(* CoDeSys 2.3.10.0 project: main.prx *)
(* Libraries: standard.lib 5.6.98 12:03:02, TcBaseBCxx50.lbx 29.3.07 07:21:36, TcSystemBCxx50.lbx 11.2.10 15:45:50 *)

(* Task configuration *)
TASK Standard (PRIORITY := 0, INTERVAL := T#20ms);
	ADS_block();
	MAIN
END_TASK

(* Global variable list: Global_Variables *)
VAR_GLOBAL
	DD1_2 AT%I* : BOOL;
	DD3  AT%I* : BOOL;
	DO1 AT%I* : BOOL;     (*не задействован*)

	DD1_2_var_off: BOOL := FALSE;
	DD1_2_var_on: BOOL := FALSE;
	DD3_var_off: BOOL := FALSE;
	DD3_var_on: BOOL := FALSE;
	delay_DD1_2_off : TIME := T#1m;
	delay_DD3_off : TIME := T#1m;

(***********out relays for landscape lights************)
	Out AT%Q* : ARRAY [1..18] OF BOOL := FALSE;

(***********out relays garage************)
	garage_OG_22_ABB_replacement AT %Q* : BOOL;
	OutLight1 AT%Q* :BOOL;     (*не задействована*)
	OutLight2 AT%Q* :BOOL;     (*не задействована*)
	OutLight3 AT%Q* :BOOL;     (*не задействована*)
	OutLight4 AT%Q* :BOOL;     (*не задействована*)

(***********keypad buttons************)
	UOG18_1 AT%I* : BOOL;	(*Клавиша ручного вкл/выкл освещения гаража в комнате охраны*)
	UOG18_2 AT%I* : BOOL;	(*Клавиша ручного вкл/выкл освещения ландшафта в комнате охраны*)
	UOG18_1_mem : BOOL;	(*положение клавиши предыдущего цикла*)
	UOG18_2_mem : BOOL;	(*положение клавиши предыдущего цикла*)
(***********keypad buttons************)

	KNX_NIGHT : BOOL;
	NIGHT_KNXNET : BOOL;
	NIGHT_KNXNET_FLAG : BOOL;
	NIGHT_CLOCK : BOOL;
	daynightbit : INT := 8;
	SystemTime : TIMESTRUCT;

	KNX_NIGHT_front: BOOL;
	KNX_DAY_front: BOOL := TRUE;
	KNX_GatesLight : BOOL;
	SWAP_CYCLE : BOOL;
	garage_OG_22 : BOOL;

	AdsUdpOutcomingStack : ARRAY [1..19] OF BOOL;
	AdsUdpReceiveStack : ARRAY [1..19] OF BOOL;
	AdsUdpEmptyStack : ARRAY [1..19] OF BOOL := FALSE;
	TESTneeds : BOOL;

	var1 : BOOL;
	var2 : BOOL;
END_VAR

(* Global variable list: TwinCAT_Configuration *)
(* Generated automatically by TwinCAT - (read only) *)
VAR_CONFIG
	.DD1_2 AT %IX8.0 : BOOL;	(*  ~ {LinkedWith:TIID^Device 1 (BX-BK)^BX KBus-Device^Term 2 (KL1408)^Channel 5^Input} *)
	.DD3 AT %IX8.1 : BOOL;	(*  ~ {LinkedWith:TIID^Device 1 (BX-BK)^BX KBus-Device^Term 2 (KL1408)^Channel 7^Input} *)
	.DO1 AT %IX8.2 : BOOL;	(*  ~ {LinkedWith:TIID^Device 1 (BX-BK)^BX KBus-Device^Term 2 (KL1408)^Channel 1^Input} *)
	.Out AT %QB4 : ARRAY [1..18] OF BOOL;
	.garage_OG_22_ABB_replacement AT %QX24.0 : BOOL;
	.OutLight1 AT %QX2.0 : BOOL;	(*  ~ {LinkedWith:TIID^Device 1 (BX-BK)^BX KBus-Device^Term 8 (KM2604)^Channel 3^Output} *)
	.OutLight2 AT %QX2.1 : BOOL;	(*  ~ {LinkedWith:TIID^Device 1 (BX-BK)^BX KBus-Device^Term 8 (KM2604)^Channel 4^Output} *)
	.OutLight3 AT %QX2.2 : BOOL;
	.OutLight4 AT %QX2.3 : BOOL;
	.UOG18_1 AT %IX12.0 : BOOL;	(*  ~ {LinkedWith:TIID^Device 1 (BX-BK)^BX KBus-Device^Term 2 (KL1408)^Channel 4^Input} *)
	.UOG18_2 AT %IX12.1 : BOOL;	(*  ~ {LinkedWith:TIID^Device 1 (BX-BK)^BX KBus-Device^Term 2 (KL1408)^Channel 2^Input} *)
END_VAR

(* POU ADS_block, CFC *)
PROGRAM ADS_block
VAR
	Timer1: TON;
	ADSreadcxbc1: ADSREAD;
	ADSreadcxbc2: ADSREAD;
	ADSwritecxbc1: ADSWRITE;
	ADSreadcxbc3: ADSREAD;
	ADSreadcxbc4: ADSREAD;
	ADSreadcxbc5: ADSREAD;
	ADSreadcxbc6: ADSREAD;
END_VAR
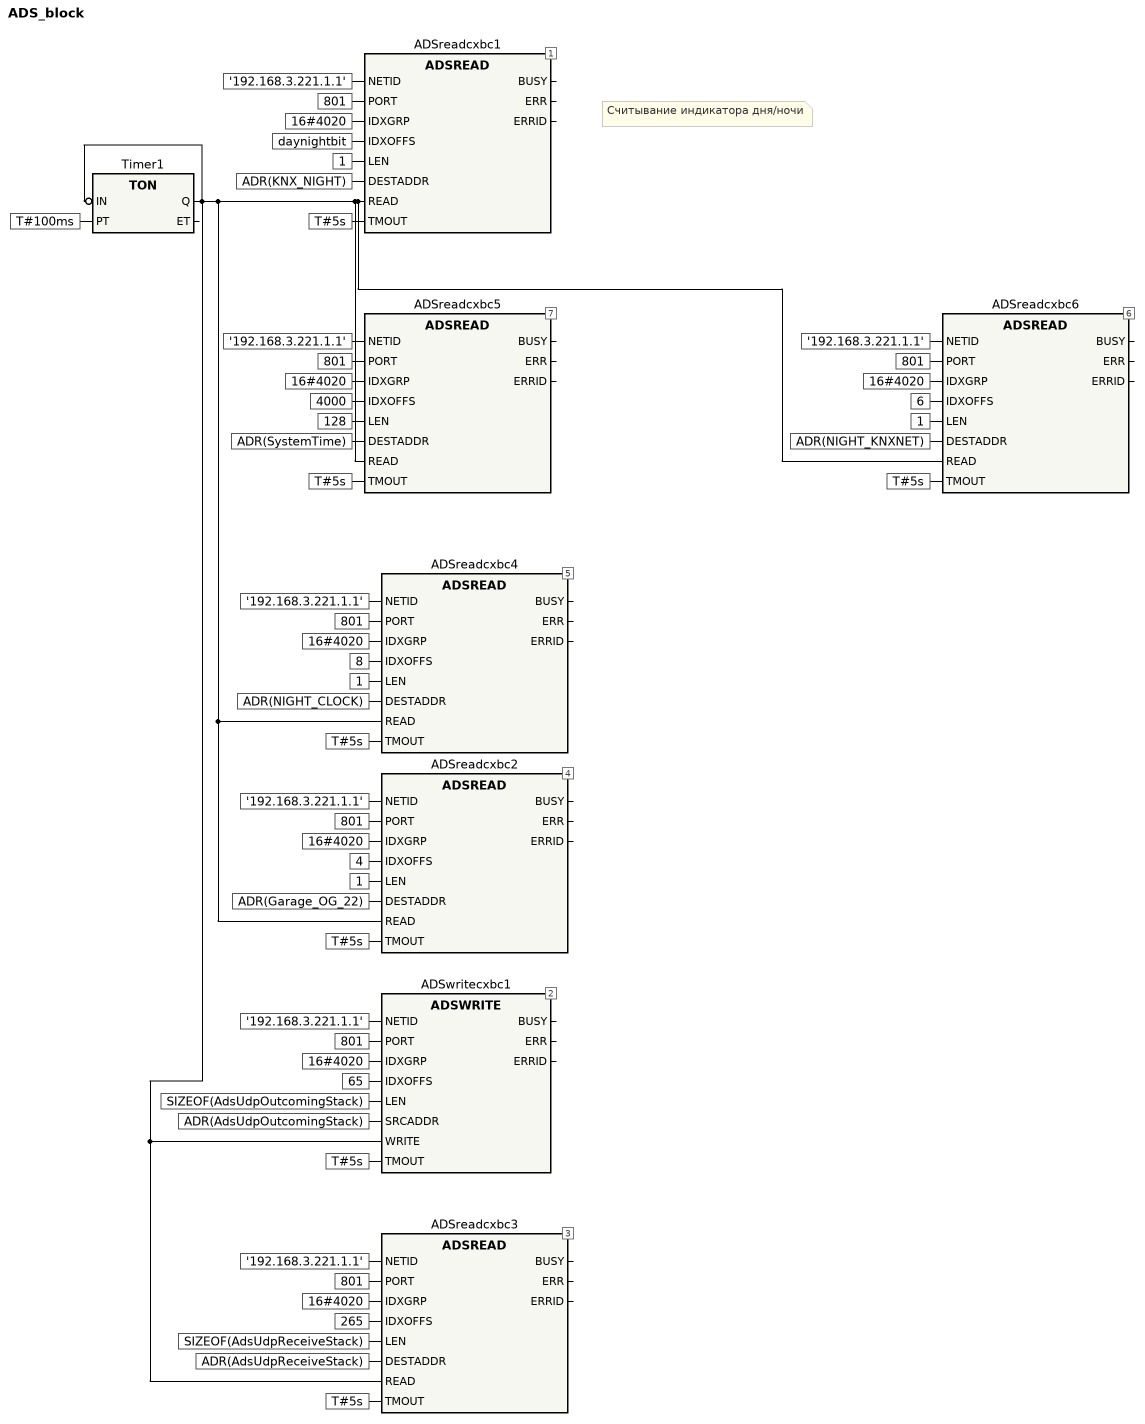
_CFC_ (* Continuous Function Chart, elements in execution order *)
#0 Timer1:TON(IN: NOT #0.Q, PT: T#100ms)
#1 ADSreadcxbc1:ADSREAD(NETID: '192.168.3.221.1.1', PORT: 801, IDXGRP: 16#4020, IDXOFFS: daynightbit, LEN: 1, DESTADDR: ADR(KNX_NIGHT), READ: #0.Q, TMOUT: T#5s)
(* Считывание индикатора дня/ночи *)
#2 ADSwritecxbc1:ADSWRITE(NETID: '192.168.3.221.1.1', PORT: 801, IDXGRP: 16#4020, IDXOFFS: 65, LEN: SIZEOF(AdsUdpOutcomingStack), SRCADDR: ADR(AdsUdpOutcomingStack), WRITE: #0.Q, TMOUT: T#5s)
#3 ADSreadcxbc3:ADSREAD(NETID: '192.168.3.221.1.1', PORT: 801, IDXGRP: 16#4020, IDXOFFS: 265, LEN: SIZEOF(AdsUdpReceiveStack), DESTADDR: ADR(AdsUdpReceiveStack), READ: #0.Q, TMOUT: T#5s)
#4 ADSreadcxbc2:ADSREAD(NETID: '192.168.3.221.1.1', PORT: 801, IDXGRP: 16#4020, IDXOFFS: 4, LEN: 1, DESTADDR: ADR(Garage_OG_22), READ: #0.Q, TMOUT: T#5s)
#5 ADSreadcxbc4:ADSREAD(NETID: '192.168.3.221.1.1', PORT: 801, IDXGRP: 16#4020, IDXOFFS: 8, LEN: 1, DESTADDR: ADR(NIGHT_CLOCK), READ: #0.Q, TMOUT: T#5s)
#6 ADSreadcxbc6:ADSREAD(NETID: '192.168.3.221.1.1', PORT: 801, IDXGRP: 16#4020, IDXOFFS: 6, LEN: 1, DESTADDR: ADR(NIGHT_KNXNET), READ: #0.Q, TMOUT: T#5s)
#7 ADSreadcxbc5:ADSREAD(NETID: '192.168.3.221.1.1', PORT: 801, IDXGRP: 16#4020, IDXOFFS: 4000, LEN: 128, DESTADDR: ADR(SystemTime), READ: #0.Q, TMOUT: T#5s)
_END_CFC_
(* the same logic as Structured Text *)
Timer1(IN := NOT Timer1.Q, PT := T#100ms);
ADSreadcxbc1(NETID := '192.168.3.221.1.1', PORT := 801, IDXGRP := 16#4020, IDXOFFS := daynightbit, LEN := 1, DESTADDR := ADR(KNX_NIGHT), READ := Timer1.Q, TMOUT := T#5s);
(* Считывание индикатора дня/ночи *)
ADSwritecxbc1(NETID := '192.168.3.221.1.1', PORT := 801, IDXGRP := 16#4020, IDXOFFS := 65, LEN := SIZEOF(AdsUdpOutcomingStack), SRCADDR := ADR(AdsUdpOutcomingStack), WRITE := Timer1.Q, TMOUT := T#5s);
ADSreadcxbc3(NETID := '192.168.3.221.1.1', PORT := 801, IDXGRP := 16#4020, IDXOFFS := 265, LEN := SIZEOF(AdsUdpReceiveStack), DESTADDR := ADR(AdsUdpReceiveStack), READ := Timer1.Q, TMOUT := T#5s);
ADSreadcxbc2(NETID := '192.168.3.221.1.1', PORT := 801, IDXGRP := 16#4020, IDXOFFS := 4, LEN := 1, DESTADDR := ADR(Garage_OG_22), READ := Timer1.Q, TMOUT := T#5s);
ADSreadcxbc4(NETID := '192.168.3.221.1.1', PORT := 801, IDXGRP := 16#4020, IDXOFFS := 8, LEN := 1, DESTADDR := ADR(NIGHT_CLOCK), READ := Timer1.Q, TMOUT := T#5s);
ADSreadcxbc6(NETID := '192.168.3.221.1.1', PORT := 801, IDXGRP := 16#4020, IDXOFFS := 6, LEN := 1, DESTADDR := ADR(NIGHT_KNXNET), READ := Timer1.Q, TMOUT := T#5s);
ADSreadcxbc5(NETID := '192.168.3.221.1.1', PORT := 801, IDXGRP := 16#4020, IDXOFFS := 4000, LEN := 128, DESTADDR := ADR(SystemTime), READ := Timer1.Q, TMOUT := T#5s);
END_PROGRAM

(* POU MAIN, ST *)
PROGRAM MAIN
VAR
	i : INT;
	FLAG_I : BOOL := TRUE;
	j: INT;
	Rec_Not_Empty: BOOL;
	k: INT;
	FLAG_01: BOOL;
	HOUR_01: WORD := 2;
	MINUTE_01: WORD := 59;
	HOUR_02: WORD := 10;
	MINUTE_02: WORD := 20;
END_VAR
IF (FLAG_I) THEN (*первый "холостой" цикл, запись положения клавиши ручного вкл/выкл освещения*)
	UOG18_1_mem := UOG18_1;
	UOG18_2_mem := UOG18_2;
	KNX_DAY_front := TRUE;
	FLAG_I := FALSE;
END_IF;

IF (Garage_OG_22) THEN
garage_OG_22_ABB_replacement := TRUE;
ELSE
garage_OG_22_ABB_replacement := FALSE;
END_IF;

IF(UOG18_1 = UOG18_1_mem) THEN; (*вкл/выкл подсветки гаража в комнате охраны*)
ELSE
	Out[5] := NOT(Out[5]);
	Out[6] := NOT(Out[6]);
END_IF;

KNX_night_init; (*подпрограмма получения флага ночь/день по фронтам переменной KNX_NIGHT*)
DD_delay_block; (*подпрограмма обработки сигнала с ДД*)
IF(UOG18_2 = UOG18_2_mem) THEN
		IF (DD1_2_var_on AND DD1_2_var_off = FALSE) THEN   (*Включение/выключение подсветки въезда в гараж от ДД*)
			Out[1] := TRUE;
		END_IF;
		IF (DD1_2_var_off AND DD1_2_var_on = FALSE) THEN
			Out[1] := FALSE;
		END_IF;
		IF (DD3_var_on AND DD3_var_off = FALSE) THEN   (*Включение/выключение подсветки дверей в электрощитовую, ДГУ от ДД*)
			Out[2] := TRUE;
		END_IF;
		IF (DD3_var_off AND DD3_var_on = FALSE) THEN
			Out[2] := FALSE;
		END_IF;
ELSE
	SWAP_CYCLE := FALSE;
	Light_Swap;
END_IF;

UOG18_1_mem := UOG18_1;
UOG18_2_mem := UOG18_2;

(*тестирование автозамены переменной дня-ночи с каэникс на временнУю*)

IF SystemTime.wHour = HOUR_01 AND SystemTime.wMinute = MINUTE_01 THEN
	FLAG_01 := NIGHT_KNXNET_FLAG;
END_IF;

IF SystemTime.wHour = HOUR_02 AND SystemTime.wMinute = MINUTE_02 AND FLAG_01 = NIGHT_KNXNET_FLAG THEN
	daynightbit := 8;
END_IF;

IF FLAG_01 = NOT(NIGHT_KNXNET_FLAG) THEN
	daynightbit := 6;
END_IF;


IF (KNX_NIGHT_front) THEN (*включение ночью*)
(* отключил для того, чтобы отдать управление AMX
	Out[3] := TRUE;
	Out[4] := FALSE;
	Out[7] := TRUE;
	Out[8] := FALSE;
	Out[9] := TRUE;
	Out[10] := FALSE;
	Out[11] := TRUE;
	Out[12] := FALSE;
	Out[13] := TRUE;
	Out[14] := FALSE;
	Out[15] := TRUE;
	Out[16] := FALSE;
	Out[17] := TRUE;
	Out[18] := FALSE; 
*)
KNX_NIGHT_front := FALSE;
END_IF;
IF (KNX_DAY_front) THEN (*выключение днем*)
(*
	Out[1] := FALSE;
	Out[2] := FALSE;
	Out[3] := FALSE;
	Out[4] := TRUE;
	Out[7] := FALSE;
	Out[8] := TRUE;
	Out[9] := FALSE;
	Out[10] := TRUE;
	Out[11] := FALSE;
	Out[12] := TRUE;
	Out[13] := FALSE;
	Out[14] := TRUE;
	Out[15] := FALSE;
	Out[16] := TRUE;
	Out[17] := FALSE;
	Out[18] := TRUE; *)
KNX_DAY_front := FALSE;
END_IF;

ADS_send_init;

Rec_Not_Empty := FALSE;

FOR k := 4 TO 17 DO
IF (AdsUdpReceiveStack[k] = AdsUdpEmptyStack[k]) THEN
Rec_Not_Empty := (Rec_Not_Empty OR FALSE);
ELSE
Rec_Not_Empty := (Rec_Not_Empty OR TRUE);
END_IF;
END_FOR;

IF (Rec_Not_Empty) THEN
Out[3] := AdsUdpReceiveStack[6];
Out[4] := NOT(AdsUdpReceiveStack[6]);
Out[5] := AdsUdpReceiveStack[7];
Out[6] := AdsUdpReceiveStack[8];
Out[7] := AdsUdpReceiveStack[9];
Out[8] := NOT(AdsUdpReceiveStack[9]);
Out[9] := AdsUdpReceiveStack[10];
Out[10] := NOT(AdsUdpReceiveStack[10]);
Out[11] := AdsUdpReceiveStack[11];
Out[12] := NOT(AdsUdpReceiveStack[11]);
Out[13] := AdsUdpReceiveStack[12];
Out[14] := NOT(AdsUdpReceiveStack[12]);
Out[15] := AdsUdpReceiveStack[13];
Out[16] := NOT(AdsUdpReceiveStack[13]);
Out[17] := AdsUdpReceiveStack[14];
Out[18] := NOT(AdsUdpReceiveStack[14]);
OutLight1 := AdsUdpReceiveStack[15];
OutLight2 := NOT(AdsUdpReceiveStack[16]);
OutLight3 := AdsUdpReceiveStack[16];
OutLight4 := AdsUdpReceiveStack[17];

AdsUdpOutcomingStack[4] := AdsUdpReceiveStack[4];
AdsUdpOutcomingStack[5] := AdsUdpReceiveStack[5];
AdsUdpOutcomingStack[6] := AdsUdpReceiveStack[6];
AdsUdpOutcomingStack[7] := AdsUdpReceiveStack[7];
AdsUdpOutcomingStack[8] := AdsUdpReceiveStack[8];
AdsUdpOutcomingStack[9] := AdsUdpReceiveStack[9];
AdsUdpOutcomingStack[10] := AdsUdpReceiveStack[10];
AdsUdpOutcomingStack[11] := AdsUdpReceiveStack[11];
AdsUdpOutcomingStack[12] := AdsUdpReceiveStack[12];
AdsUdpOutcomingStack[13] := AdsUdpReceiveStack[13];
AdsUdpOutcomingStack[14] := AdsUdpReceiveStack[14];
AdsUdpOutcomingStack[15] := AdsUdpReceiveStack[15];
AdsUdpOutcomingStack[16] := AdsUdpReceiveStack[16];
AdsUdpOutcomingStack[17] := AdsUdpReceiveStack[17];

AdsUdpEmptyStack := AdsUdpReceiveStack;
END_IF;
IF(TESTneeds) THEN AdsUdpReceiveStack := AdsUdpOutcomingStack; END_IF;
END_PROGRAM

(* POU KNX_night_init, ST *)
PROGRAM KNX_night_init
VAR
	Rising_edge_trig1 : R_TRIG;
	Falling_edge_trig1 : F_TRIG;

	Rising_edge_trig2 : R_TRIG;
	Falling_edge_trig2 : F_TRIG;
END_VAR
Rising_edge_trig1 (CLK := KNX_NIGHT, Q => );
IF (Rising_edge_trig1.Q) THEN
	KNX_NIGHT_front := TRUE;
END_IF;
Falling_edge_trig1 (CLK := KNX_NIGHT, Q => );
IF (Falling_edge_trig1.Q) THEN
	KNX_DAY_front := TRUE;
	DD1_2_var_off := TRUE;
	DD1_2_var_on := FALSE;
	DD3_var_off := TRUE;
	DD3_var_on := FALSE;
END_IF;

Rising_edge_trig2 (CLK := NIGHT_KNXNET, Q => );
Falling_edge_trig2 (CLK := NIGHT_KNXNET, Q => );
IF (Rising_edge_trig2.Q OR Falling_edge_trig2.Q) THEN
	NIGHT_KNXNET_FLAG := NOT(NIGHT_KNXNET_FLAG);
END_IF;
END_PROGRAM

(* POU DD_delay_block, CFC *)
PROGRAM DD_delay_block
VAR
	Timer1_2 : TON;
	Timer3 : TON;
	TP01: TP;
	TP02: TP;
	TP03: TP;
	TP04: TP;
	TP05: TP;
	TP06: TP;
	TP07: TP;
	TP08: TP;
END_VAR
VAR (* helpers for the ST form of the networks *)
	_t65 : BOOL;
	_t84 : BOOL;
	_t121 : BOOL;
	_t132 : BOOL;
END_VAR
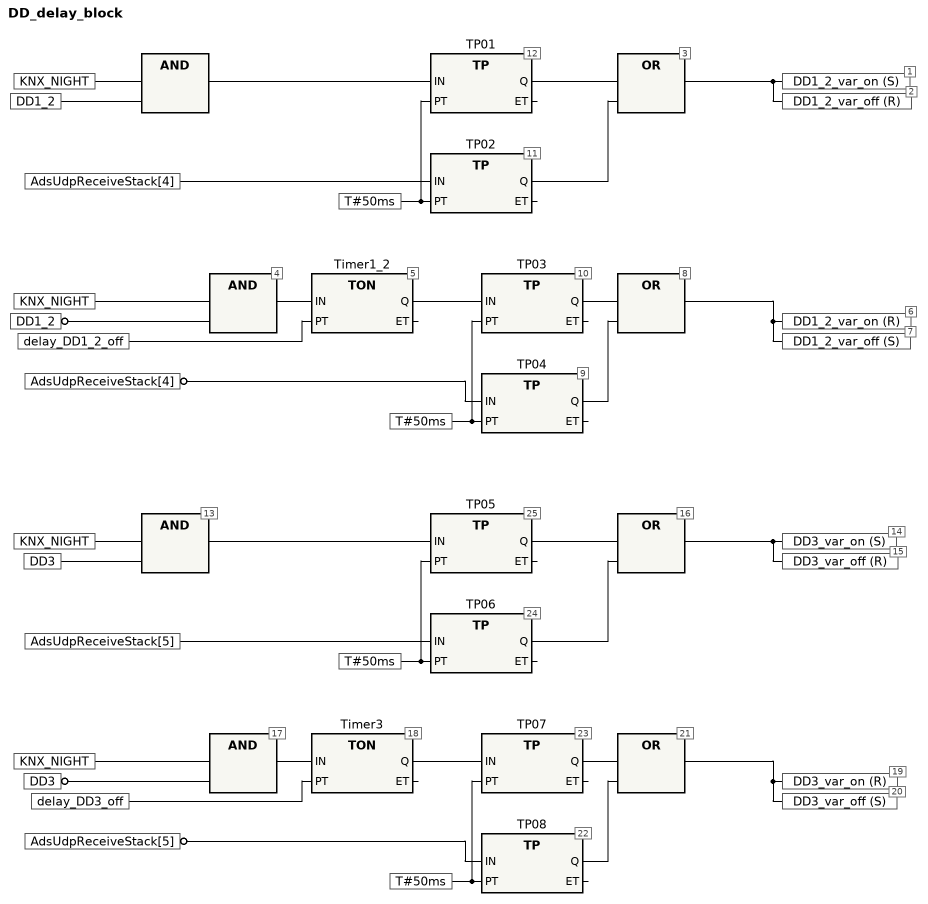
_CFC_ (* Continuous Function Chart, elements in execution order *)
#0 AND(KNX_NIGHT, DD1_2)
#1 S DD1_2_var_on <= #3
#2 R DD1_2_var_off <= #3
#3 OR(#12.Q, #11.Q)
#4 AND(KNX_NIGHT, NOT DD1_2)
#5 Timer1_2:TON(IN: #4, PT: delay_DD1_2_off)
#6 R DD1_2_var_on <= #8
#7 S DD1_2_var_off <= #8
#8 OR(#10.Q, #9.Q)
#9 TP04:TP(IN: NOT AdsUdpReceiveStack[4], PT: T#50ms)
#10 TP03:TP(IN: #5.Q, PT: T#50ms)
#11 TP02:TP(IN: AdsUdpReceiveStack[4], PT: T#50ms)
#12 TP01:TP(IN: #0, PT: T#50ms)
#13 AND(KNX_NIGHT, DD3)
#14 S DD3_var_on <= #16
#15 R DD3_var_off <= #16
#16 OR(#25.Q, #24.Q)
#17 AND(KNX_NIGHT, NOT DD3)
#18 Timer3:TON(IN: #17, PT: delay_DD3_off)
#19 R DD3_var_on <= #21
#20 S DD3_var_off <= #21
#21 OR(#23.Q, #22.Q)
#22 TP08:TP(IN: NOT AdsUdpReceiveStack[5], PT: T#50ms)
#23 TP07:TP(IN: #18.Q, PT: T#50ms)
#24 TP06:TP(IN: AdsUdpReceiveStack[5], PT: T#50ms)
#25 TP05:TP(IN: #13, PT: T#50ms)
_END_CFC_
(* the same logic as Structured Text *)
IF _t65 THEN DD1_2_var_on := TRUE; END_IF;
IF _t65 THEN DD1_2_var_off := FALSE; END_IF;
_t65 := TP01.Q OR TP02.Q;
Timer1_2(IN := KNX_NIGHT AND NOT DD1_2, PT := delay_DD1_2_off);
IF _t84 THEN DD1_2_var_on := FALSE; END_IF;
IF _t84 THEN DD1_2_var_off := TRUE; END_IF;
_t84 := TP03.Q OR TP04.Q;
TP04(IN := NOT AdsUdpReceiveStack[4], PT := T#50ms);
TP03(IN := Timer1_2.Q, PT := T#50ms);
TP02(IN := AdsUdpReceiveStack[4], PT := T#50ms);
TP01(IN := KNX_NIGHT AND DD1_2, PT := T#50ms);
IF _t121 THEN DD3_var_on := TRUE; END_IF;
IF _t121 THEN DD3_var_off := FALSE; END_IF;
_t121 := TP05.Q OR TP06.Q;
Timer3(IN := KNX_NIGHT AND NOT DD3, PT := delay_DD3_off);
IF _t132 THEN DD3_var_on := FALSE; END_IF;
IF _t132 THEN DD3_var_off := TRUE; END_IF;
_t132 := TP07.Q OR TP08.Q;
TP08(IN := NOT AdsUdpReceiveStack[5], PT := T#50ms);
TP07(IN := Timer3.Q, PT := T#50ms);
TP06(IN := AdsUdpReceiveStack[5], PT := T#50ms);
TP05(IN := KNX_NIGHT AND DD3, PT := T#50ms);
END_PROGRAM

(* POU Light_Swap, ST *)
PROGRAM Light_Swap
VAR
END_VAR
IF ((Out[3] OR Out[7] OR Out[9] OR Out[1] OR Out[13] OR Out[15] OR Out[17]) AND SWAP_CYCLE = FALSE) THEN (*если горит хотя бы один из ландшафтных светильников, то выключаем ВСЕ: ландшафтные и наружное освещение гаража*)
	Out[1] := FALSE;
	Out[2] := FALSE;
	Out[3] := FALSE;
	Out[4] := TRUE;
	Out[7] := FALSE;
	Out[8] := TRUE;
	Out[9] := FALSE;
	Out[10] := TRUE;
	Out[11] := FALSE;
	Out[12] := TRUE;
	Out[13] := FALSE;
	Out[14] := TRUE;
	Out[15] := FALSE;
	Out[16] := TRUE;
	Out[17] := FALSE;
	Out[18] := TRUE;
	KNX_NIGHT_front := FALSE; (*при переключении клавиши отключаем флаг ночи, чтобы воспрепятствовать автоматическому включению света (ночью). Отныне свет управляется только с этой клавиши вручную. Автоматическая работа алгоритма возобновится с очередным передним фронтом переменной KNX_NIGHT*)
	SWAP_CYCLE := TRUE; (*индикатор срабатывания свапа [воизбежание зацикливания подпрограммы]*)
END_IF;
IF ((Out[4] OR Out[8] OR Out[10] OR Out[12] OR Out[14] OR Out[16] OR Out[18]) AND SWAP_CYCLE = FALSE) THEN (*если не горит хотя бы один из ландшафтных светильников, то включаем ВСЕ: ландшафтные и наружное освещение гаража*)
	Out[1] := TRUE;
	Out[2] := TRUE;
	Out[3] := TRUE;
	Out[4] := FALSE;
	Out[7] := TRUE;
	Out[8] := FALSE;
	Out[9] := TRUE;
	Out[10] := FALSE;
	Out[11] := TRUE;
	Out[12] := FALSE;
	Out[13] := TRUE;
	Out[14] := FALSE;
	Out[15] := TRUE;
	Out[16] := FALSE;
	Out[17] := TRUE;
	Out[18] := FALSE;
	KNX_NIGHT_front := TRUE; (*при переключении клавиши включаем флаг ночи, чтобы воспрепятствовать автоматическому выключению света (днём). Отныне свет управляется только с этой клавиши вручную. Автоматическая работа алгоритма возобновится с очередным задним фронтом переменной KNX_NIGHT*)
	SWAP_CYCLE := TRUE; (*индикатор срабатывания свапа [воизбежание зацикливания подпрограммы]*)
END_IF;
END_PROGRAM

(* POU ADS_send_init, ST *)
PROGRAM ADS_send_init
VAR
END_VAR
AdsUdpOutcomingStack[1] := DD1_2;
AdsUdpOutcomingStack[2] := DD3;
AdsUdpOutcomingStack[3] := DO1;
AdsUdpOutcomingStack[4] := Out[1];
AdsUdpOutcomingStack[5] := Out[2];
AdsUdpOutcomingStack[6] := Out[3];
AdsUdpOutcomingStack[7] := Out[5];
AdsUdpOutcomingStack[8] := Out[6];
AdsUdpOutcomingStack[9] := Out[7];
AdsUdpOutcomingStack[10] := Out[9];
AdsUdpOutcomingStack[11] := Out[11];
AdsUdpOutcomingStack[12] := Out[13];
AdsUdpOutcomingStack[13] := Out[15];
AdsUdpOutcomingStack[14] := Out[17];
AdsUdpOutcomingStack[15] := OutLight1;
AdsUdpOutcomingStack[16] := OutLight3;
AdsUdpOutcomingStack[17] := OutLight4;
AdsUdpOutcomingStack[18] := UOG18_1;
AdsUdpOutcomingStack[19] := UOG18_2;
END_PROGRAM

(* Visualisation Test
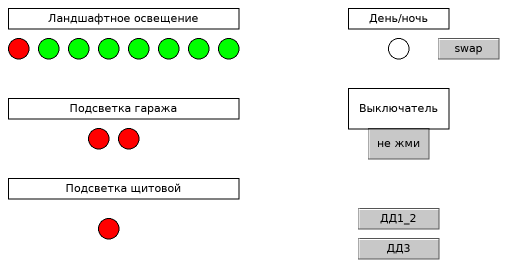
ellipse at (160,50)-(181,71): invisible if Out[3]
ellipse at (160,50)-(181,71): invisible if Out[4]
rectangle at (130,20)-(361,41): text "Ландшафтное освещение"
ellipse at (190,50)-(211,71): invisible if Out[7]
ellipse at (190,50)-(211,71): invisible if Out[8]
ellipse at (220,50)-(241,71): invisible if Out[9]
ellipse at (220,50)-(241,71): invisible if Out[10]
ellipse at (250,50)-(271,71): invisible if Out[11]
ellipse at (250,50)-(271,71): invisible if Out[12]
ellipse at (280,50)-(301,71): invisible if Out[13]
ellipse at (280,50)-(301,71): invisible if Out[14]
ellipse at (310,50)-(331,71): invisible if Out[15]
ellipse at (310,50)-(331,71): invisible if Out[16]
ellipse at (340,50)-(361,71): invisible if Out[17]
ellipse at (340,50)-(361,71): invisible if Out[18]
button at (490,140)-(551,171): text "не жми"; toggles UOG18
ellipse at (510,50)-(531,71): alarm colour if KNX_NIGHT
rectangle at (470,20)-(571,41): text "День/ночь"
rectangle at (470,100)-(571,141): text "Выключатель"
button at (480,220)-(561,241): text "ДД1_2"; taps DD1_2
button at (480,250)-(561,271): text "ДД3"; taps DD3
ellipse at (130,50)-(151,71): alarm colour if Out[6]
ellipse at (210,140)-(231,161): alarm colour if Out[1]
rectangle at (130,110)-(361,131): text "Подсветка гаража"
ellipse at (240,140)-(261,161): alarm colour if Out[5]
rectangle at (130,190)-(361,211): text "Подсветка щитовой"
ellipse at (220,230)-(241,251): alarm colour if Out[2]
button at (560,50)-(621,71): text "swap"; toggles KNX_NIGHT
*)
